// TwinCAT 3 PLC project PLC
// ProgramVersion: 3.1.4023.0
// libraries:
//   Tc2_Standard, * (Beckhoff Automation GmbH)
//   Tc2_System, * (Beckhoff Automation GmbH)
//   Tc3_Module, * (Beckhoff Automation GmbH)
// project tree:
//   DUTs/ stBelt.TcDUT, stCmd.TcDUT, stOB.TcDUT
//   GVLs/ OPCUA.TcGVL
//   / PlcTask.TcTTO
//   POUs/ MAIN.TcPOU
// real-time tasks:
//   TASK PlcTask: cycle T#10ms, priority 20, ADS port 350
// I/O:
//   DEVICE Dispositivo 1 (EtherCAT) (disabled), AmsNetId 192.168.2.41.2.1
//     Terminale 1 (EK1200) [EK1200-5000 EtherCAT Power supply (2A E-Bus)]
//       Terminale 2 (EL9100) [EL9100 Power Supplier with LED (24V)]
//       Terminale 8 (EL1819) [EL1819 16Ch. Dig. Input 24V, 10µs]
//       Terminale 7 (EL1819) [EL1819 16Ch. Dig. Input 24V, 10µs]
//       Terminale 9 (EL2809) [EL2809 16Ch. Dig. Output 24V, 0.5A]
//       Terminale 10 (EL6224-0090) [EL6224-0090 (IO Link Master, TwinSAFE SC)]
//         modules: Module 1 (DeviceState Inputs Device), Module 2 (DeviceState Inputs), Module 3 (IO-Link Slave), Module 4 (empty), Module 5 (empty), Module 6 (empty)
//       Terminale 11 (EK1122) [EK1122 2 port EtherCAT junction]
//         Terminale 12 (EK1100) [EK1100 EtherCAT Coupler (2A E-Bus)]
//           Terminale 24 (EL1018) [EL1018 8Ch. Dig. Input 24V, 10µs]
//           Terminale 14 (EL6224-0090) [EL6224-0090 (IO Link Master, TwinSAFE SC)]
//             modules: Module 1 (DeviceState Inputs Device), Module 2 (DeviceState Inputs), Module 3 (IO-Link Slave), Module 4 (IO-Link Slave), Module 5 (IO-Link Slave), Module 6 (empty)
//           Terminale 15 (EL6224-0090) [EL6224-0090 (IO Link Master, TwinSAFE SC)]
//             modules: Module 1 (DeviceState Inputs Device), Module 2 (DeviceState Inputs), Module 3 (empty), Module 4 (empty), Module 5 (empty), Module 6 (empty)
//           Terminale 16 (EL6224-0090) [EL6224-0090 (IO Link Master, TwinSAFE SC)]
//             modules: Module 1 (DeviceState Inputs Device), Module 2 (DeviceState Inputs), Module 3 (empty), Module 4 (empty), Module 5 (empty), Module 6 (empty)
//           Terminale 17 (EL6224-0090) [EL6224-0090 (IO Link Master, TwinSAFE SC)]
//             modules: Module 1 (DeviceState Inputs Device), Module 2 (DeviceState Inputs), Module 3 (empty), Module 4 (empty), Module 5 (empty), Module 6 (empty)
//           Terminale 18 (EL6224-0090) [EL6224-0090 (IO Link Master, TwinSAFE SC)]
//             modules: Module 1 (DeviceState Inputs Device), Module 2 (DeviceState Inputs), Module 3 (empty), Module 4 (empty), Module 5 (empty), Module 6 (empty)
//           Terminale 25 (EL9011) [EL9011 End Terminal]
//         Terminale 13 (EK1100) [EK1100 EtherCAT Coupler (2A E-Bus)]
//           Terminale 19 (EL6224-0090) [EL6224-0090 (IO Link Master, TwinSAFE SC)]
//             modules: Module 1 (DeviceState Inputs Device), Module 2 (DeviceState Inputs), Module 3 (empty), Module 4 (empty), Module 5 (empty), Module 6 (empty)
//           Terminale 20 (EL6224-0090) [EL6224-0090 (IO Link Master, TwinSAFE SC)]
//             modules: Module 1 (DeviceState Inputs Device), Module 2 (DeviceState Inputs), Module 3 (empty), Module 4 (empty), Module 5 (empty), Module 6 (empty)
//           Terminale 21 (EL6224-0090) [EL6224-0090 (IO Link Master, TwinSAFE SC)]
//             modules: Module 1 (DeviceState Inputs Device), Module 2 (DeviceState Inputs), Module 3 (empty), Module 4 (empty), Module 5 (empty), Module 6 (empty)
//           Terminale 22 (EL6224-0090) [EL6224-0090 (IO Link Master, TwinSAFE SC)]
//             modules: Module 1 (DeviceState Inputs Device), Module 2 (DeviceState Inputs), Module 3 (empty), Module 4 (empty), Module 5 (empty), Module 6 (empty)
//           Terminale 23 (EL6224-0090) [EL6224-0090 (IO Link Master, TwinSAFE SC)]
//             modules: Module 1 (DeviceState Inputs Device), Module 2 (DeviceState Inputs), Module 3 (empty), Module 4 (empty), Module 5 (empty), Module 6 (empty)
//           Terminale 26 (EL9011) [EL9011 End Terminal]
//       Terminale 3 (EK1122) [EK1122 2 port EtherCAT junction]
//         N. box 4 (INVT_ECAT_100) [INVT_ECAT_100]
//         101 [INVT_ECAT_100]
//         101_1 [INVT_ECAT_100]
//         101_2 [INVT_ECAT_100]
//         101_3 [INVT_ECAT_100]
//         101_4 [INVT_ECAT_100]
//         101_5 [INVT_ECAT_100]
//         101_6 [INVT_ECAT_100]
//         101_7 [INVT_ECAT_100]
//         101_8 [INVT_ECAT_100]
//         101_9 [INVT_ECAT_100]
//         N. box 5 (MultiControl EtherCAT) [MultiControl EtherCAT]
//       Terminale 6 (EL9011) [EL9011 End Terminal]

CONFIGURATION PLC
    RESOURCE PLC ON TwinCAT3
        TASK PlcTask(INTERVAL := T#10ms, PRIORITY := 20);
        PROGRAM MAIN WITH PlcTask : MAIN;
    END_RESOURCE
END_CONFIGURATION

// ---- DUTs/stBelt.TcDUT
{attribute 'OPC.UA.DA.StructuredType' := '1'}
TYPE stBelt :
STRUCT
	sName		: STRING[10];
	uliOrder	: ULINT;
	xFull		: BOOL;
	xEmpty		: BOOL;
	xAvailable	: BOOL;
	xEnable		: BOOL;
END_STRUCT
END_TYPE

// ---- DUTs/stCmd.TcDUT
{attribute 'OPC.UA.DA.StructuredType' := '1'}
TYPE stCmd :
STRUCT
	iCmd	: INT;	(* Codice comando *)
	iPar1	: INT;	(* Parametro 1 *)
	iPar2	: INT;	(* Parametro 2 *)
END_STRUCT
END_TYPE

// ---- DUTs/stOB.TcDUT
{attribute 'OPC.UA.DA.StructuredType' := '1'}
TYPE stOB :
STRUCT
	sName		: STRING[10];
	uliOrder	: ULINT;
	xFull		: BOOL;
	xEmpty		: BOOL;
	xAvailable	: BOOL;
	xEnable		: BOOL;
END_STRUCT
END_TYPE

// ---- GVLs/OPCUA.TcGVL

VAR_GLOBAL
	{attribute 'OPC.UA.DA' := '1'}	
	aOBN1		: ARRAY[0..20] OF stOB;		(* Array buffer su nastro 1 *)
	{attribute 'OPC.UA.DA' := '1'}
	aOBN2		: ARRAY[0..20] OF stOB;		(* Array buffer su nastro 2 *)
	{attribute 'OPC.UA.DA' := '1'}	
	aOBN3		: ARRAY[0..20] OF stOB;		(* Array buffer su nastro 3 *)
	{attribute 'OPC.UA.DA' := '1'}	
	aNastri_L1	: ARRAY[0..5] OF stBelt;	(* Array nastri linea 1 *)
	{attribute 'OPC.UA.DA' := '1'}	
	aNastri_L2	: ARRAY[0..5] OF stBelt;	(* Array nastri linea 2) *)
	{attribute 'OPC.UA.DA' := '1'}	
	CmdNastro1Linea1	: stCmd;	(* Comandi per nastro 1 Linea 1 *) 
	{attribute 'OPC.UA.DA' := '1'}	
	CmdNastro2Linea1	: stCmd;	(* Comandi per nastro 2 Linea 1 *) 
	{attribute 'OPC.UA.DA' := '1'}	
	CmdNastro3Linea1	: stCmd;	(* Comandi per nastro 3 Linea 1 *) 
	{attribute 'OPC.UA.DA' := '1'}	
	CmdNastro4Linea1	: stCmd;	(* Comandi per nastro 4 Linea 1 *) 
	{attribute 'OPC.UA.DA' := '1'}	
	CmdNastro1Linea2	: stCmd;	(* Comandi per nastro 1 Linea 2 *) 
	{attribute 'OPC.UA.DA' := '1'}	
	CmdNastro2Linea2	: stCmd;	(* Comandi per nastro 2 Linea 2 *) 
	{attribute 'OPC.UA.DA' := '1'}	
	CmdNastro3Linea2	: stCmd;	(* Comandi per nastro 3 Linea 2 *) 
	{attribute 'OPC.UA.DA' := '1'}	
	CmdNastro4Linea2	: stCmd;	(* Comandi per nastro 4 Linea 2 *) 
	{attribute 'OPC.UA.DA' := '1'}	
	CmdObFinale			: StCmd;	(* Comandi per OB fine linea *)

END_VAR

// ---- POUs/MAIN.TcPOU
PROGRAM MAIN
VAR
END_VAR

END_PROGRAM
